// TIA Portal V20 export
TYPE "OEM_Data"
// stored: Access Published, Namespace CITI_Logic
   STRUCT
      Assistance_Call : Array[1..8] of Bool;
      Assistance_CallAck : Array[1..8] of Bool;
      OUT_TL_Call : Bool;
      PMC : "CITI_Logic.PMC_Input_Data";
      CITI_OneShot { S7_SetPoint := 'True'} : Array[1..32] of Bool;
      System_Byte : Byte;
      FirstScan : Bool;
      Always_OFF : Bool;
      Always_ON : Bool;
      DiagStatusUpdate : Bool;
      Clock_Byte : Byte;
      ClockMemByte_Example : Byte;
      Null_String : String;
      TO_COMPLETE : Bool;
      TO_COMPLETE_INT : Int;
      RESERVED : Byte;
      MachineFaultedLevel1 : Bool;
      MachineFaultedLevel2 : Bool;
      FaultString : String[200];
      Empty_Pallet : Bool;
      OUT_ShiftNumber : Byte;
      OUT_Flasher : Bool;
      LampCheck : Bool;
      Red_Light : Bool;
      Green_Light : Bool;
      Blue_Light : Bool;
      Yellow_Light : Bool;
      No_Maps_Have_Fault_Delay : IEC_TIMER;
      IN_Fault_String_Null { S7_SetPoint := 'True'} : Bool;
      Fault_String_is_Null : Bool;
      FlexNet : "CITI_Logic.FlexNet_Data";
      FlexNet_Response_Fault_Count { S7_SetPoint := 'True'} : Int;
      FlexNet_No_Response_Fault : Bool;
      FlexNet_No_Response_Warning : Bool;
      FlexNet_Transaction_Retry_Occurred : Bool;
      FlexNet_DataReceivedByHost : Bool;
      FlexNet_Response_FLT_Time : S5Time;
   END_STRUCT;
END_TYPE
